# B&R Automation Studio project VC4toMappView
Automation Studio 4.11.6.26 SP; technology packages: mappView 5.24.0

## Configuration Config1

CPU PC_any, AutomationRuntime D4.92, Build 4.1.2, Vc V4.72.5

### Task classes (Cpu.sw)
```
Cyclic#1:
  Program <- Program.prg
VcDataObjects: VisuVC <- VisuVC4.dob
Binaries: vcctext, vcpfar00, vcfile, udbdef, vcpdsw, mvLoader, vcshared, vcgclass, vcmgr, vctcal, vcnet, vcpdvnc, vcdsint, vccbtn, VisuVC01, vcalarm, VisuVC02, FWRules, vcpkat, vcrt, TCData, vcbclass, vcfntttf, vcdsloc, arial, ashwac, User, sysconf, asfw, arconfig, ashwd, iomap, Role
Libraries: arssl, astime, asieccon, runtime, fileio, vcresman, dataobj
```

### Hardware
```
PC : PC_any v1.1.1.0 (OrderNumber=PC)
  Connector IF3:
    Vnc1
    VncVcObjectName1 = VisuVC
    VncKeyMappingFile1 = VC\PS2-Keyboard.dis
    VncMaxConnections1 = 4
  ConfigurationID = VC4toMappView_Config1
  FileDevice1
  FileDeviceName1 = USER
  FileDevicePath1 = USER_PATH
```

## Logical view

- Visualisation Logical/mappView (not shown)

- Visualisation Logical/VisuVC4 (not shown)

### Program Logical/Program (IEC)

#### Variables.var
```iecst
VAR
	Boo : BOOL;
END_VAR
```

#### Main.st
```iecst
PROGRAM _INIT
	(* Insert code here *)

END_PROGRAM

PROGRAM _CYCLIC
	(* Insert code here *)
	 Boo;
END_PROGRAM

PROGRAM _EXIT
	(* Insert code here *)

END_PROGRAM
```

Listed in the project but not available here: Logical/Global.typ, Logical/Global.var, Logical/Libraries
